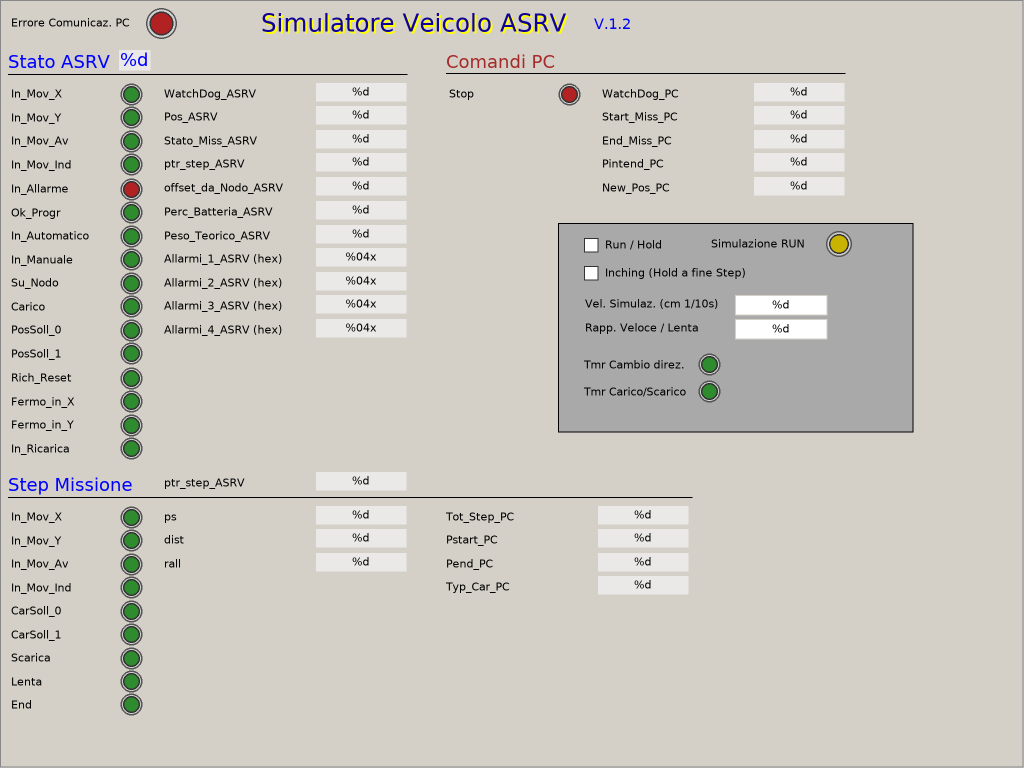
VISUALIZATION Visualization  // 1024x768
    Rectangle (558,223 355x209)
    Label (8,79 113x30), "In_Mov_X"
    Label (8,103 113x30), "In_Mov_Y"
    Lamp1 (119,82 25x25), variable: sSta.Stato_ASRV.In_Mov_X, style: Lamp-Lamp1-Green
    Lamp1 (119,105 25x25), variable: sSta.Stato_ASRV.In_Mov_Y, style: Lamp-Lamp1-Green
    Label (8,126 113x30), "In_Mov_Av"
    Label (8,150 113x30), "In_Mov_Ind"
    Lamp1 (119,129 25x25), variable: sSta.Stato_ASRV.In_Mov_Av, style: Lamp-Lamp1-Green
    Lamp1 (119,152 25x25), variable: sSta.Stato_ASRV.In_Mov_Ind, style: Lamp-Lamp1-Green
    Label (8,174 113x30), "In_Allarme"
    Label (8,198 113x30), "Ok_Progr"
    Lamp1 (119,177 25x25), variable: sSta.Stato_ASRV.In_Allarme, style: Lamp-Lamp1-Red
    Lamp1 (119,200 25x25), variable: sSta.Stato_ASRV.Ok_Prog, style: Lamp-Lamp1-Green
    Label (8,221 113x30), "In_Automatico"
    Label (8,245 113x30), "In_Manuale"
    Lamp1 (119,224 25x25), variable: sSta.Stato_ASRV.In_Automatico, style: Lamp-Lamp1-Green
    Lamp1 (119,247 25x25), variable: sSta.Stato_ASRV.In_Manuale, style: Lamp-Lamp1-Green
    Label (8,268 113x30), "Su_Nodo"
    Label (8,292 113x30), "Carico"
    Lamp1 (119,271 25x25), variable: sSta.Stato_ASRV.Su_Nodo, style: Lamp-Lamp1-Green
    Lamp1 (119,294 25x25), variable: sSta.Stato_ASRV.Carico, style: Lamp-Lamp1-Green
    Label (8,315 113x30), "PosSoll_0"
    Label (8,339 113x30), "PosSoll_1"
    Lamp1 (119,318 25x25), variable: sSta.Stato_ASRV.PosSoll_0, style: Lamp-Lamp1-Green
    Lamp1 (119,341 25x25), variable: sSta.Stato_ASRV.PosSoll_1, style: Lamp-Lamp1-Green
    Label (8,363 113x30), "Rich_Reset"
    Label (8,387 113x30), "Fermo_in_X"
    Lamp1 (119,366 25x25), variable: sSta.Stato_ASRV.Rich_Reset, style: Lamp-Lamp1-Green
    Lamp1 (119,389 25x25), variable: sSta.Stato_Aux_ASRV.Fermo_in_X, style: Lamp-Lamp1-Green
    Label (8,410 113x30), "Fermo_in_Y"
    Label (8,434 113x30), "In_Ricarica"
    Lamp1 (119,413 25x25), variable: sSta.Stato_Aux_ASRV.Fermo_in_Y, style: Lamp-Lamp1-Green
    Lamp1 (119,436 25x25), variable: sSta.Stato_Aux_ASRV.In_Ricarica, style: Lamp-Lamp1-Green
    Label (8,8 132x30), "Errore Comunicaz. PC"
    Lamp1 (144,6 35x35), variable: bErrComPc, style: Lamp-Lamp1-Red
    Label (5,47 143x30), "Stato ASRV"
    Label (161,102 130x30), "Pos_ASRV"
    Label (161,126 130x30), "Stato_Miss_ASRV"
    Label (161,149 130x30), "ptr_step_ASRV"
    Label (161,173 130x30), "offset_da_Nodo_ASRV"
    Label (161,197 130x30), "Perc_Batteria_ASRV"
    Label (161,221 130x30), "Peso_Teorico_ASRV"
    Label (161,244 130x30), "Allarmi_1_ASRV (hex)"
    Label (161,268 130x30), "Allarmi_2_ASRV (hex)"
    Label (161,291 130x30), "Allarmi_3_ASRV (hex)"
    Label (161,315 130x30), "Allarmi_4_ASRV (hex)"
    Textfield (315,105 92x20), "%d", text variable: sTxSta.Pos_ASRV
    Textfield (315,129 92x20), "%d", text variable: sTxSta.Stato_Miss_ASRV
    Textfield (315,152 92x20), "%d", text variable: sTxSta.ptr_step_ASRV
    Textfield (315,176 92x20), "%d", text variable: sTxSta.offset_da_nodo_ASRV
    Textfield (315,200 92x20), "%d", text variable: sTxSta.Perc_Batteria_ASRV
    Textfield (315,224 92x20), "%d", text variable: sTxSta.Peso_Teorico_ASRV
    Textfield (315,247 92x20), "%04x", text variable: sTxSta.Allarmi_1_ASRV
    Textfield (315,271 92x20), "%04x", text variable: sTxSta.Allarmi_2_ASRV
    Textfield (315,294 92x20), "%04x", text variable: sTxSta.Allarmi_3_ASRV
    Textfield (315,318 92x20), "%04x", text variable: sTxSta.Allarmi_4_ASRV
    Label (161,79 130x30), "WatchDog_ASRV"
    Textfield (315,82 92x20), "%d", text variable: sTxSta.WatchDog_ASRV
    Label (446,79 113x30), "Stop"
    Lamp1 (557,82 25x25), variable: fbClassAsrv.sAsrv.ASRV_CMD.Comando_PC.Stop, style: Lamp-Lamp1-Red
    Label (443,47 143x30), "Comandi PC"
    Label (599,102 130x30), "Start_Miss_PC"
    Label (599,126 130x30), "End_Miss_PC"
    Label (599,149 130x30), "Pintend_PC"
    Label (599,173 130x30), "New_Pos_PC"
    Textfield (753,105 92x20), "%d", text variable: sRxCmd.Start_Miss_PC
    Textfield (753,129 92x20), "%d", text variable: sRxCmd.End_Miss_PC
    Textfield (753,152 92x20), "%d", text variable: sRxCmd.Pintend_PC
    Textfield (753,176 92x20), "%d", text variable: sRxCmd.New_Pos_PC
    Label (599,79 130x30), "WatchDog_PC"
    Textfield (753,82 92x20), "%d", text variable: sRxCmd.WatchDog_PC
    Line (8,74) (407,74)
    Line (446,73) (845,73)
    Label (8,502 113x30), "In_Mov_X"
    Label (8,526 113x30), "In_Mov_Y"
    Lamp1 (119,505 25x25), variable: sLastStep.Comandi.In_Mov_X, style: Lamp-Lamp1-Green
    Lamp1 (119,528 25x25), variable: sLastStep.Comandi.In_Mov_Y, style: Lamp-Lamp1-Green
    Label (8,549 113x30), "In_Mov_Av"
    Label (8,573 113x30), "In_Mov_Ind"
    Lamp1 (119,552 25x25), variable: sLastStep.Comandi.In_Mov_Av, style: Lamp-Lamp1-Green
    Lamp1 (119,575 25x25), variable: sLastStep.Comandi.In_Mov_Ind, style: Lamp-Lamp1-Green
    Label (5,470 143x30), "Step Missione"
    Label (161,525 130x30), "dist"
    Label (161,549 130x30), "rall"
    Textfield (315,528 92x20), "%d", text variable: sLastStep.dist
    Textfield (315,552 92x20), "%d", text variable: sLastStep.rall
    Label (161,502 130x30), "ps"
    Textfield (315,505 92x20), "%d", text variable: sLastStep.ps
    Line (8,497) (692,497)
    Label (8,596 113x30), "CarSoll_0"
    Label (8,620 113x30), "CarSoll_1"
    Lamp1 (119,599 25x25), variable: sLastStep.Comandi.CarSoll_0, style: Lamp-Lamp1-Green
    Lamp1 (119,622 25x25), variable: sLastStep.Comandi.CarSoll_1, style: Lamp-Lamp1-Green
    Label (8,643 113x30), "Scarica"
    Label (8,667 113x30), "Lenta"
    Lamp1 (119,646 25x25), variable: sLastStep.Comandi.Scarica, style: Lamp-Lamp1-Green
    Lamp1 (119,669 25x25), variable: sLastStep.Comandi.Lenta, style: Lamp-Lamp1-Green
    Label (161,468 130x30), "ptr_step_ASRV"
    Textfield (315,471 92x20), "%d", text variable: sTxSta.ptr_step_ASRV
    Label (8,690 113x30), "End"
    Lamp1 (119,692 25x25), variable: sLastStep.Comandi.End, style: Lamp-Lamp1-Green
    Label (443,525 130x30), "Pstart_PC"
    Label (443,549 130x30), "Pend_PC"
    Label (443,572 130x30), "Typ_Car_PC"
    Textfield (597,528 92x20), "%d", text variable: fbClassAsrv.sAsrv.ASRV_MIS.Pstart_PC
    Textfield (597,552 92x20), "%d", text variable: fbClassAsrv.sAsrv.ASRV_MIS.Pend_PC
    Textfield (597,575 92x20), "%d", text variable: fbClassAsrv.sAsrv.ASRV_MIS.Typ_car_PC
    Label (443,502 130x30), "Tot_Step_PC"
    Textfield (597,505 92x20), "%d", text variable: fbClassAsrv.sAsrv.ASRV_MIS.Tot_step_PC
    Textfield (118,49 33x22), "%d", text variable: fbClassAsrv.sAsrv.ASRV_num
    Label (582,289 150x30), "Vel. Simulaz. (cm 1/10s)"
    Textfield (735,295 92x20), "%d", text variable: nSimCmSpost
        OnMouseClick: write the text variable via VisuDialogs.Numpad, min 1, max 100
    Label (582,313 150x30), "Rapp. Veloce / Lenta"
    Textfield (735,319 92x20), "%d", text variable: nRappVelLen
        OnMouseClick: write the text variable via VisuDialogs.Numpad, min 1, max 20
    Label (708,229 113x30), "Simulazione RUN"
    Lamp1 (824,229 30x30), variable: bSimulaRun, style: Lamp-Lamp1-Yellow
    Label (581,350 113x30), "Tmr Cambio direz."
    Lamp1 (697,352 25x25), variable: bCambioDir, style: Lamp-Lamp1-Green
    Label (260,10 330x30), "Simulatore Veicolo ASRV"
    Label (258,8 330x30), "Simulatore Veicolo ASRV"
    Label (591,9 49x30), "V.1.2"
    Checkbox (582,230 103x30), "Run / Hold", variable: bSimulaRun
    Checkbox (582,258 201x30), "Inching (Hold a fine Step)", variable: bSimulaStep
    Label (581,377 113x30), "Tmr Carico/Scarico"
    Lamp1 (697,379 25x25), variable: bCarScar, style: Lamp-Lamp1-Green
END_VISUALIZATION

(* stored: Version 1.1.0.1, ProductVersion 3.1.4024.11
   Visu Visualization: Id {758707e3-0ff7-47e2-be11-ce156cb9633e} *)
